	    //Dispatchers value
	    // GRIPPER/ROBOT NEL REFRESH (5/10, concordato 24/7): era l'unico one-shot
	    // che il 90 non ripubblicava. Va accodato DOPO i 32 DISPATCH: il refresh
	    // ne inserisce piu' di quanti il buffer d'invio (11 posti, circolare) ne
	    // tenga, e sopravvivono solo gli ultimi. Il 90 mette Dispatcher_old a -1:
	    // lo si annota in #temp prima che il FOR lo riallinei.
	    #temp := 0;
	    IF #Dispatcher_old[31] = -1 THEN
	        #temp := 1;
	    END_IF;
	    FOR #i := 0 TO 31 DO
	        IF #Dispatcher_old[#i] <> #Dispatcher[#i] THEN
	            "FC_MQTT"(insert := true,
	                      send := false,
	                      topic := CONCAT(IN1 := 'FROM_PLANT/DISPATCH/ROBOT/', IN2 := "INT_TO_STRING_WITHOUT_SIGN"(#i)),
	                      payload := STRING_TO_WSTRING("INT_TO_STRING_WITHOUT_SIGN"(#Dispatcher[#i])));

	            #Dispatcher_old[#i] := #Dispatcher[#i];
	        END_IF;
	    END_FOR;
	    IF #temp = 1 THEN
	        "FC_MQTT"(insert := true,
	                  send := false,
	                  topic := 'FROM_PLANT/GRIPPER/ROBOT',
	                  payload := STRING_TO_WSTRING("INT_TO_STRING_WITHOUT_SIGN"(#Gripper_ID[1])));
	    END_IF;

	END_REGION

	REGION resetDispatcher
	    (*IF NOT #RemoteMode OR ("DB_MQTT".lastTopicReceived = 'ROBOT' AND "DB_MQTT".lastCmdReceived > "CMD_RobotReset") THEN*)
	    IF #RESET_ALL_DISPATCH OR "Start_AUX" OR "ResetAreaRobot" THEN
	        #Dispatcher["_master"] := 0;
	        #Dispatcher["_Pallet_TRAY_to_Robot"] := 0;
	        #Dispatcher["_Pallet_Robot_to_TRAY"] := 0;
	        #Dispatcher["_Pallet_Robot_to_MC"] := 0;
	        #Dispatcher["_Pallet_MC_to_Robot"] := 0;
	        #Dispatcher["_Part_TRAY_to_Robot"] := 0;
	        #Dispatcher["_Part_Robot_to_TRAY"] := 0;
	        #Dispatcher["_Part_Robot_to_MC"] := 0;
	        #Dispatcher["_Part_MC_to_Robot"] := 0;
	        #Dispatcher["_Set_Gripper_OnBoard"] := 0;   // ex _Vice_TRAY_to_Robot (17/9)
	        #Dispatcher["_Vice_Robot_to_TRAY"] := 0;
	        #Dispatcher["_Vice_Robot_to_MC"] := 0;
	        #Dispatcher["_Vice_MC_to_Robot"] := 0;
	        #Dispatcher["_Gripper_TRAY_to_Robot"] := 0;
	        #Dispatcher["_Gripper_Robot_to_TRAY"] := 0;
	        #Dispatcher["_Gripper_Hook_Search"] := 0;
	        #Dispatcher["_Gripper4Pallet_Search"] := 0;
	        #Dispatcher["updatePartOnTray"] := 0;
	        #Dispatcher["Extract_TRAY"] := 0;
	        #Dispatcher["Release_TRAY"] := 0;
	        #Dispatcher["change_TCP_Data"] := 0;
	        #Dispatcher["get_TCP_Data"] := 0;
	        #Dispatcher["updateGripperOnRobot"] := 0;
	        #Dispatcher["updatePartOnRobot"] := 0;
	        #Dispatcher["updatePartOnMC"] := 0;
	        #Dispatcher["updatePalletOnTRAY"] := 0;
	        #Dispatcher["Extract_TRAY_HMI"] := 0;
	        #Dispatcher["Release_TRAY_HMI"] := 0;
	        #Dispatcher["executeOneQuery"] := 0;
	        #Dispatcher["Reset_or_log_MissionData"] := 0;
	        #Dispatcher["_Declare_Position"] := 0;
	        #retryPick := FALSE;
	        "DB_executeQuery".readyForNextQuery := TRUE;
	        #queryStartExecution := false;

	        // Il ponte SQL va liberato COMPLETAMENTE: azzerando le catene senza
	        // questo, FB6 resta fermo allo stato 35 in attesa di un chiamante che
	        // non esiste piu' e sqlCommands[0] non si svuota mai -> tutta la cella
	        // si blocca in silenzio.
	        "DB_executeQuery".Dispatch["_master"] := 0;
	        "SqlCommands".sqlCommands[0] := '';
	        #queryTemp := '';


	        // consensi spinta in battuta: se restano alti dopo un reset, il robot
	        // li legge come validi alla missione successiva
	        "Q_PushEnable_MC" := FALSE;
	        "Ok_PushSpinta_MC" := FALSE;
	        "Ok_PushArrivo_MC" := FALSE;
	        // e il consenso di fase 2 della missione 16 (5/10): stesso motivo
	        "Ok_Phase2_MC" := FALSE;

	        // COMANDO MANUALE CON FB204 IN CICLO (5/10). I comandi manuali in HOLD
	        // (home, posizionamenti, restart programma) e la dichiarazione 35 azzerano
	        // le catene e MissionCode senza errore: FB204, fermo ad aspettare una
	        // missione, leggeva "MissionCode = 0" come missione riuscita e andava
	        // avanti (es. 57 -> 58 -> ricetta e start con la morsa vuota).
	        // Il reset robot (99) e AUX riportano gia' FB204 a 0 (qui il master e'
	        // gia' 0 per il 99, e AUX lo azzera piu' sotto). Per gli altri comandi:
	        //   - stati di attesa missione fuori lavorazione (lista della guardia D2
	        //     di FB204 senza il 95): 9999 con allarme 959, si riparte dal pannello
	        //     dopo aver dichiarato lo stato della cella;
	        //   - 95 (HAAS in lavorazione): non si abbandona il ciclo macchina, si
	        //     salta al substate 6 e si aspetta la fine ciclo;
	        //   - tutti gli altri stati restano dove sono.
	        // Si ritira la query prenotata di FB204 (il ponte e' appena stato
	        // svuotato) ma NON queryTemp: il rilevamento "query persa" di FB204 la
	        // rifa' da solo.
	        IF #RESET_ALL_DISPATCH AND "DB_MC1".Dispatcher["_master"] <> 0 THEN
	            IF "DB_MC1".Dispatcher["_master"] = 95 THEN
	                "DB_MC1".subState := 6;
	            ELSIF ("DB_MC1".Dispatcher["_master"] = 30 AND ("DB_MC1".subState = 1 OR "DB_MC1".subState = 2))
	                OR "DB_MC1".Dispatcher["_master"] = 35
	                OR "DB_MC1".Dispatcher["_master"] = 43
	                OR "DB_MC1".Dispatcher["_master"] = 44
	                OR "DB_MC1".Dispatcher["_master"] = 46
	                OR ("DB_MC1".Dispatcher["_master"] >= 50 AND "DB_MC1".Dispatcher["_master"] <= 59)
	                OR "DB_MC1".Dispatcher["_master"] = 96
	                OR "DB_MC1".Dispatcher["_master"] = 965
	                OR "DB_MC1".Dispatcher["_master"] = 966
	                OR ("DB_MC1".Dispatcher["_master"] >= 103 AND "DB_MC1".Dispatcher["_master"] <= 105)
	            THEN
	                "FC_MQTT"(insert := true,
	               send := false,
	               topic := 'FROM_PLANT/ALARM/MC1',
	               payload := STRING_TO_WSTRING('959'));   // ciclo interrotto da comando manuale
	                "DB_MC1".io_out.startWork := FALSE;
	                "DB_MC1".Dispatcher["_master"] := 9999;
	            END_IF;
	            "DB_MC1".queryStartExecution := FALSE;
	        END_IF;

	        #RESET_ALL_DISPATCH := FALSE;

	        #swapDataReady := FALSE;
	    END_IF;

	    IF "Start_AUX" OR "ResetAreaRobot" THEN
	        "DB_RobotMission".Command := 0;
	        "DB_MC1".Dispatcher["_master"] := 0;
	        "DB_MC2".Dispatcher["_master"] := 0;
	        #MissionCode := 0;
	        #swapDataReady := FALSE;
	    END_IF;

	END_REGION

	REGION PLANT STATUS FOR ROBOT
	    IF #MCRequested = 1 THEN
	        "DB_RobotMission".cmd_Status.DoorClosed := NOT "DB_MC1".io_in.doorOpened;
	    END_IF;
	END_REGION

	REGION Supervisione coerenza pinza
	    // INIBITA DURANTE LA DICHIARAZIONE (18/9): dopo un reinit i registri sono
	    // a zero con la pinza fisicamente a bordo — la condizione e' vera per
	    // costruzione e il timer scade prima che l'operatore riesca a dichiarare.
	    // Il comando 35 azzera #Error, ma tonCoerenza.Q e' gia' alto e lo rialza
	    // nello stesso scan: il pannello vede l'errore e rifiuta la sequenza.
	    // Finche' il Declare_State sta lavorando, l'incoerenza e' ATTESA: e' proprio
	    // quello che si sta correggendo.
	    #tonCoerenza(IN := "DB_RobotMissionStatus".StatusCode = "cmd_waitingNewCmd"
	                 AND #Dispatcher["_Declare_State"] = 0
	                 AND ("Gripper_mounted" XOR (#Gripper_ID[1] > 0)),
	                 PT := T#2s);
	    IF #tonCoerenza.Q AND #Error = 0 THEN
	        #Error := 938;
	    END_IF;
	END_REGION

	REGION Publish sensori pinza
	    IF BOOL_TO_INT("Gripper_mounted") <> #mounted_old THEN
	        "FC_MQTT"(insert := true,
	                  send := false,
	                  topic := 'FROM_PLANT/GRIPPER/MOUNTED',
	                  payload := STRING_TO_WSTRING("INT_TO_STRING_WITHOUT_SIGN"(BOOL_TO_INT("Gripper_mounted"))));
	        #mounted_old := BOOL_TO_INT("Gripper_mounted");
	    END_IF;
	    IF BOOL_TO_INT("Gripper1_Closed") <> #closed1_old THEN
	        "FC_MQTT"(insert := true,
	                  send := false,
	                  topic := 'FROM_PLANT/GRIPPER/CLOSED1',
	                  payload := STRING_TO_WSTRING("INT_TO_STRING_WITHOUT_SIGN"(BOOL_TO_INT("Gripper1_Closed"))));
	        #closed1_old := BOOL_TO_INT("Gripper1_Closed");
	    END_IF;
	END_REGION


	// Sicurezza: pubblicazione CICLICA, non solo on-change.
	// Un pannello che si connette dopo, o che perde il messaggio, resterebbe con uno
	// stato di sicurezza stantio e bloccherebbe i comandi all'operatore: e' successo
	// il 3/9 e ha fermato la linea.
	//
	#tonSafetyPub(IN := NOT #tonSafetyPub.Q,
	              PT := T#3s);
	IF #tonSafetyPub.Q OR "Main_Safety_RTG1_DB".Aux_OK <> #auxOK_old THEN
	    "FC_MQTT"(insert := true,
	              send := false,
	              topic := 'FROM_PLANT/SAFETY/AUX',
	              payload := STRING_TO_WSTRING("INT_TO_STRING_WITHOUT_SIGN"(BOOL_TO_INT("Main_Safety_RTG1_DB".Aux_OK))));
	    #auxOK_old := "Main_Safety_RTG1_DB".Aux_OK;
	END_IF;

	"Q_MC1_GateClosed" := "Q_STO_Units_CH1";
END_FUNCTION_BLOCK

